RoboDK station: vision.rdk

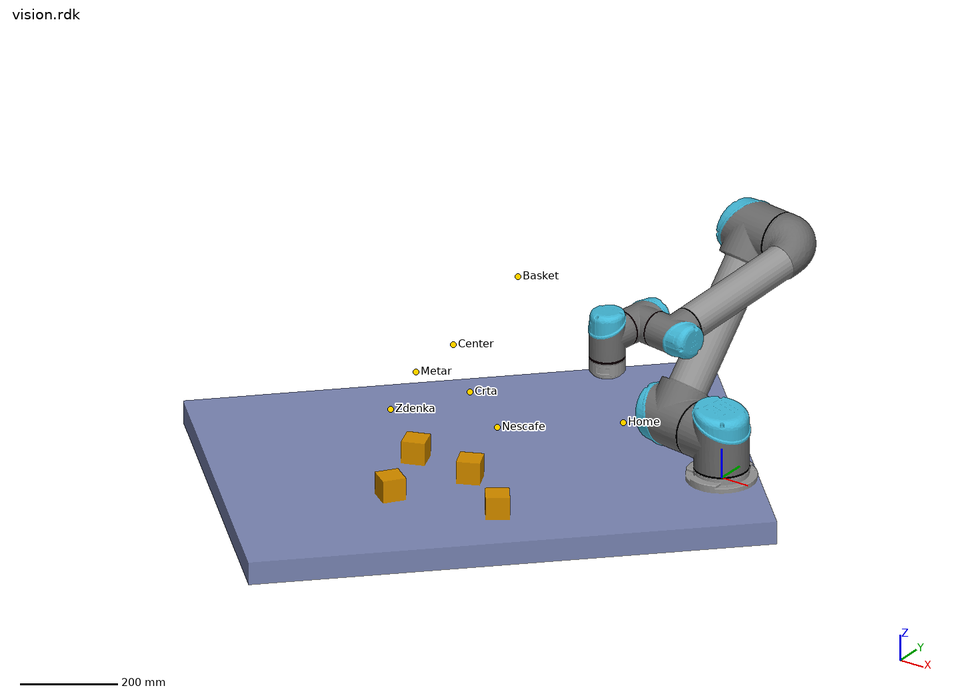
[picture v0: the station drawn from its stored meshes, robots at their saved joint values, targets as dots, program paths as lines]
Station vision (saved by RoboDK 5.5.4). Poses are relative to the parent item; angles as X-Y-Z fixed-axis rotations.
  - frame UR5 Base at (0, 0, 0) mm
    - robot UR5: 6 axes
        modified DH rows (alpha deg, a mm, theta deg, d mm): 0, 0, 0, 89.2; 90, 0, 180, 0; 0, 425, 0, 0; 0, 392, 0, 109.3; -90, 0, 0, 94.75; 90, 0, 180, 82.5
        joint limits [-360, -360, -360, -360, -360, -360] to [360, 360, 360, 360, 360, 360]; home [0, -90, -90, 0, 90, 0]; saved at [-98.231, -52.983, -136.055, -81.133, 89.967, 150.662]
    - object Zdenka at (-504.89, -461.94, 0) mm, rotated rx 0 ry 0 rz -125.23 deg, size 50 x 50 x 50 mm, geometry from Cube-50mm.sld
    - object Metar at (-562.32, -289.21, 0) mm, rotated rx 0 ry 0 rz -69.75 deg, size 50 x 50 x 50 mm, geometry from Cube-50mm.sld
    - object Nescafe at (-277.38, -404.93, 0) mm, rotated rx 0 ry 0 rz 37.42 deg, size 50 x 50 x 50 mm, geometry from Cube-50mm.sld
    - object Crta at (-417.76, -301.87, 0) mm, rotated rx 0 ry 0 rz 114.46 deg, size 50 x 50 x 50 mm, geometry from Cube-50mm.sld
    - object table at (-450, -220, -50) mm, rotated rx 90 ry 0 rz 45 deg, size 1100 x 50 x 770 mm, geometry from table.STEP
    - target Home (Cartesian target) at (-97.13, -212.15, 183.49) mm, rotated rx -179.84 ry -0.05 rz 21.11 deg; joints [-98.231, -52.983, -136.055, -81.133, 89.967, 150.662] of UR5
    - target Basket (Cartesian target) at (-516.59, 11.08, 310.25) mm, rotated rx -179.33 ry 0 rz -53.84 deg; joints [-173.806, -94.045, -88.665, -87.867, 89.663, 150.039] of UR5
    - target Center (Cartesian target) at (-450.44, -314.27, 303.64) mm, rotated rx -179.56 ry -0.63 rz 8.4 deg; joints [-137.661, -101.097, -81.602, -88.065, 89.986, 123.932] of UR5
    - target Zdenka (Cartesian target) at (-504.89, -461.94, 200) mm, rotated rx 179.99 ry 0 rz 0 deg; joints [-98.231, -52.983, -136.055, -81.133, 89.967, 150.662] of UR5
    - target Nescafe (Cartesian target) at (-277.38, -404.93, 200) mm, rotated rx 179.99 ry 0 rz 0 deg; joints [-98.231, -52.983, -136.055, -81.133, 89.967, 150.662] of UR5
    - target Metar (Cartesian target) at (-562.32, -289.21, 200) mm, rotated rx 179.99 ry 0 rz 0 deg; joints [-98.231, -52.983, -136.055, -81.133, 89.967, 150.662] of UR5
    - target Crta (Cartesian target) at (-417.76, -301.87, 200) mm, rotated rx 179.99 ry 0 rz 0 deg; joints [-98.231, -52.983, -136.055, -81.133, 89.967, 150.662] of UR5
  - program Prog1 (2 instructions, listed below)
  - Python program Prog2 (listed below)

--- program Prog1 (robot UR5) ---
  Set speed (50.0 mm/s)
  Call Prog2

--- Python program Prog2 ---
from robodk import robolink  # RoboDK API
from robodk import robodialogs  # Dialogs
from robodk.robomath import *

items = [{"item" : "Zdenka", "pic" : "test3\item3.jpg", "height" : 20},
        {"item" : "Nescafe", "pic" : "test3\item1.jpg", "height" : 65},
        {"item" : "Metar", "pic" : "test3\item4.jpg", "height" : 40},
        {"item" : "Crta", "pic" : "test3\item2.jpg", "height" : 47}]

def runmain():
    RDK = robolink.Robolink()
    RDK.setSimulationSpeed(1)
    robot = RDK.Item("UR5")
    home = RDK.Item("Home", 6)
    basket = RDK.Item("Basket",6)
    center = RDK.Item("Center",6)
    robot.MoveJ(home)

    target_dist = []

    for item in items:
        target = RDK.Item(item["item"], 6)
        pose = Pose_2_TxyzRxyz(target.Pose())
        distance = sqrt(pose[0]**2 + pose[1]**2)
        target_dist.append({"item" : item["item"], "distance" : distance, "height" : item["height"]})

    sorted_targets = sorted(target_dist, key=lambda d: d['distance'])

    for item in sorted_targets:
        target = RDK.Item(item["item"], 6)
        print(item)
        robot.MoveJ(target)
        robot.MoveL(target.Pose()*transl(0,0,200-item["height"]+30))
        robot.setDO(1, 1)
        robot.MoveL(target)
        robot.MoveJ(center)
        robot.MoveJ(basket)
        robot.setDO(1,0)
        robot.MoveJ(center)

    robot.MoveJ(home)

if __name__ == '__main__':
    runmain()
